KUKA KRL program: rob_ok.src, rob_ok.dat

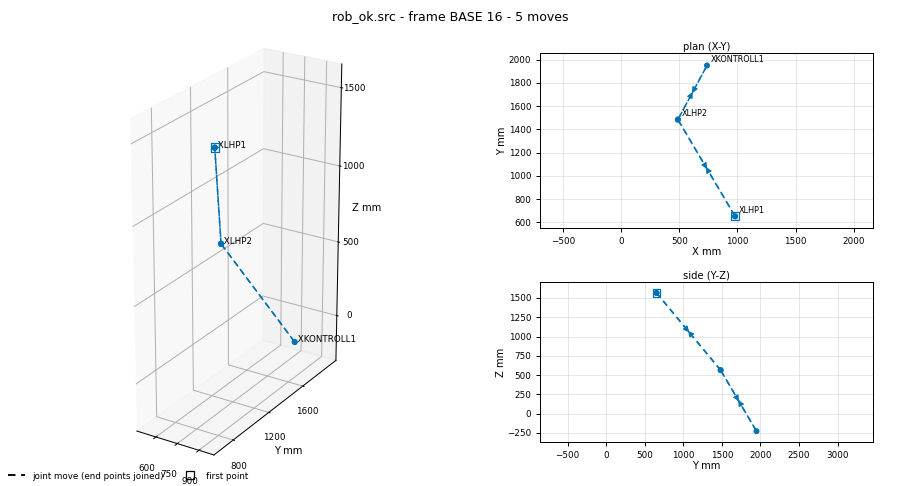
[picture p0: tool path of rob_ok.src in frame BASE 16, 5 of 7 moves have a stored position in this frame; points joined in program order, loops and branches not executed]
--- rob_ok.src ---
&ACCESS RVP
&REL 12
&COMMENT Roboterpruefprogramm
&PARAM TEMPLATE = C:\KRC\ROBOTER\TEMPLATE\VG_HP
&PARAM EDITMASK = *
DEF rob_ok( )
;FOLD INI
;FOLD BASISTECH INI
    GLOBAL INTERRUPT DECL 3 WHEN $STOPMESS==TRUE DO IR_STOPM ( )
    INTERRUPT ON 3
    BAS (#INITMOV,0 )
;ENDFOLD (BASISTECH INI)
;FOLD SPOTTECH INI
    USERSPOT(#INIT)
;ENDFOLD (SPOTTECH INI)
;FOLD GRIPPERTECH INI
    USER_GRP(0,DUMMY,DUMMY,GDEFAULT)
;ENDFOLD (GRIPPERTECH INI)
;FOLD USER INI
;Make your modifications here
;FOLD COLLISION_V_3.01 INI ;%{E}
    IF (COLLISION_DATA[1].I_NR>0) THEN
    GLOBAL INTERRUPT DECL 21 WHEN $IN[COLLISION_DATA[1].I_NR]==FALSE DO COLLSTOP (1,0 )
    ENDIF
    IF (COLLISION_DATA[2].I_NR>0) THEN
    GLOBAL INTERRUPT DECL 22 WHEN $IN[COLLISION_DATA[2].I_NR]==FALSE DO COLLSTOP (2,0 )
    ENDIF
    IF (COLLISION_DATA[3].I_NR>0) THEN
    GLOBAL INTERRUPT DECL 23 WHEN $IN[COLLISION_DATA[3].I_NR]==FALSE DO COLLSTOP (3,0 )
    ENDIF
    IF (COLLISION_DATA[4].I_NR>0) THEN
    GLOBAL INTERRUPT DECL 24 WHEN $IN[COLLISION_DATA[4].I_NR]==FALSE DO COLLSTOP (4,0 )
    ENDIF
;ENDFOLD (Collision)
;ENDFOLD (USER INI)
;ENDFOLD (INI)
;FOLD ; Anlagenbezeichn:               Stations-Nr:;%{PE}%R 5.2.7,%MKUKATPBASIS,%CCOMMENT,%VNORMAL,%P 2:Anlagenbezeichn:               Stations-Nr:
;ENDFOLD
;FOLD ; Stand / Version:;%{PE}%R 5.2.7,%MKUKATPBASIS,%CCOMMENT,%VNORMAL,%P 2:Stand / Version:
;ENDFOLD
;FOLD ; Name Bearbeiter:;%{PE}%R 5.2.7,%MKUKATPBASIS,%CCOMMENT,%VNORMAL,%P 2:Name Bearbeiter:
;ENDFOLD
;Sicherheitsfrage (nur im Musterprogramm, nach teachen entfernen)
wait for false
;FOLD ; ***************************************;%{PE}%R 2.4.6,%MKUKATPBASIS,%CCOMMENT,%VNORMAL,%P 2:***************************************
;ENDFOLD
;FOLD ; A C H T U N G  ! ! !   Nur in T1 fahren;%{PE}%R 2.4.6,%MKUKATPBASIS,%CCOMMENT,%VNORMAL,%P 2:A C H T U N G  ! ! !   Nur in T1 fahren
;ENDFOLD
;FOLD ; ***************************************;%{PE}%R 2.4.6,%MKUKATPBASIS,%CCOMMENT,%VNORMAL,%P 2:***************************************
;ENDFOLD
WAIT FOR $T1
;FOLD PTP HOME  Vel= 100 % DEFAULT;%{PE}%R 3.2.43,%MKUKATPBASIS,%CMOVE,%VPTP,%P 1:PTP, 2:HOME, 3:, 5:100, 7:DEFAULT
    $BWDSTART = FALSE
    PDAT_ACT=PDEFAULT
    BAS(#PTP_DAT)
    FDAT_ACT=FHOME
    BAS(#FRAMES)
    BAS(#VEL_PTP,100)
    $H_POS=XHOME
    PTP XHOME
;ENDFOLD
; PTP ... zur Kontrollposition Roboter teachen
;FOLD PTP LHP1  Vel= 100 % PDAT Tool[16] Base[16];%{PE}%R 3.2.43,%MKUKATPBASIS,%CMOVE,%VPTP,%P 1:PTP, 2:LHP1, 3:, 5:100, 7:PDAT
    $BWDSTART = FALSE
    PDAT_ACT=PPDAT
    BAS(#PTP_DAT)
    FDAT_ACT=FLHP1
    BAS(#FRAMES)
    BAS(#VEL_PTP,100)
    PTP XLHP1
;ENDFOLD
;FOLD PTP LHP2  Vel= 100 % PDAT Tool[16] Base[16];%{PE}%R 3.2.43,%MKUKATPBASIS,%CMOVE,%VPTP,%P 1:PTP, 2:LHP2, 3:, 5:100, 7:PDAT
    $BWDSTART = FALSE
    PDAT_ACT=PPDAT
    BAS(#PTP_DAT)
    FDAT_ACT=FLHP2
    BAS(#FRAMES)
    BAS(#VEL_PTP,100)
    PTP XLHP2
;ENDFOLD
;FOLD ; *********************************************************;%{PE}%R 2.4.6,%MKUKATPBASIS,%CCOMMENT,%VNORMAL,%P 2:*********************************************************
;ENDFOLD
;FOLD ; A C H T U N G  ! ! !   Spitze am IR Flansch befestigen   ;%{PE}%R 2.4.6,%MKUKATPBASIS,%CCOMMENT,%VNORMAL,%P 2:A C H T U N G  ! ! !   Spitze am IR Flansch befestigen
;ENDFOLD
;FOLD ; *********************************************************;%{PE}%R 2.4.6,%MKUKATPBASIS,%CCOMMENT,%VNORMAL,%P 2:*********************************************************
;ENDFOLD
;Spitze am Flansch 02.3 und 03.1
;Spitze an Vorrichtung 01.2 und 03.1
WAIT FOR  $IN[1026]==TRUE
;FOLD ; 1.Kontrollposition;%{PE}%R 2.4.6,%MKUKATPBASIS,%CCOMMENT,%VNORMAL,%P 2:1.Kontrollposition
;ENDFOLD
;FOLD ; Pruefspitze - Roboterflansch         ;%{PE}%R 2.4.6,%MKUKATPBASIS,%CCOMMENT,%VNORMAL,%P 2: Pruefspitze - Roboterflansch
;ENDFOLD
;FOLD ; mit 02.3 03.1 Laenge;%{PE}%R 5.2.17,%MKUKATPBASIS,%CCOMMENT,%VNORMAL,%P 2:mit 02.3 03.1 Laenge
;ENDFOLD
;FOLD PTP KONTROLL1  Vel= 100 % PDAT Tool[16] Base[16];%{PE}%R 3.2.43,%MKUKATPBASIS,%CMOVE,%VPTP,%P 1:PTP, 2:KONTROLL1, 3:, 5:100, 7:PDAT
    $BWDSTART = FALSE
    PDAT_ACT=PPDAT
    BAS(#PTP_DAT)
    FDAT_ACT=FKONTROLL1
    BAS(#FRAMES)
    BAS(#VEL_PTP,100)
    PTP XKONTROLL1
;ENDFOLD
WAIT FOR  $IN[1026]==TRUE ; Kontrollposition IR
;FOLD PTP LHP3  Vel= 100 % PDAT Tool[16] Base[16];%{PE}%R 3.2.43,%MKUKATPBASIS,%CMOVE,%VPTP,%P 1:PTP, 2:LHP3, 3:, 5:100, 7:PDAT
    $BWDSTART = FALSE
    PDAT_ACT=PPDAT
    BAS(#PTP_DAT)
    FDAT_ACT=FLHP3
    BAS(#FRAMES)
    BAS(#VEL_PTP,100)
    PTP XLHP3
;ENDFOLD
;FOLD ; *******************************************************;%{PE}%R 2.4.6,%MKUKATPBASIS,%CCOMMENT,%VNORMAL,%P 2:*******************************************************
;ENDFOLD
;FOLD ; A C H T U N G  ! ! !   Messpitze am IR  entfernen;%{PE}%R 2.4.6,%MKUKATPBASIS,%CCOMMENT,%VNORMAL,%P 2:A C H T U N G  ! ! !   Messpitze am IR  entferne
;ENDFOLD
;FOLD ; *******************************************************;%{PE}%R 2.4.6,%MKUKATPBASIS,%CCOMMENT,%VNORMAL,%P 2:*******************************************************
;ENDFOLD
WAIT FOR  $IN[1026]==TRUE
;FOLD PTP LHP5  Vel= 100 % PDAT Tool[16] Base[16];%{PE}%R 3.2.43,%MKUKATPBASIS,%CMOVE,%VPTP,%P 1:PTP, 2:LHP5, 3:, 5:100, 7:PDAT
    $BWDSTART = FALSE
    PDAT_ACT=PPDAT
    BAS(#PTP_DAT)
    FDAT_ACT=FLHP5
    BAS(#FRAMES)
    BAS(#VEL_PTP,100)
    PTP XLHP5
;ENDFOLD
;FOLD PTP HOME  Vel= 100 % DEFAULT;%{PE}%R 3.2.43,%MKUKATPBASIS,%CMOVE,%VPTP,%P 1:PTP, 2:HOME, 3:, 5:100, 7:DEFAULT
    $BWDSTART = FALSE
    PDAT_ACT=PDEFAULT
    BAS(#PTP_DAT)
    FDAT_ACT=FHOME
    BAS(#FRAMES)
    BAS(#VEL_PTP,100)
    $H_POS=XHOME
    PTP XHOME
;ENDFOLD
END

--- rob_ok.dat ---
&ACCESS RVP
&REL 12
&COMMENT Roboterpruefprogramm
&PARAM TEMPLATE = C:\KRC\ROBOTER\TEMPLATE\VG_HP
&PARAM EDITMASK = *
DEFDAT  ROB_OK
;FOLD EXTERNAL DECLARATIONS;%{PE}%V3.2.0,%MKUKATPBASIS,%CEXT,%VCOMMON,%P
;ENDFOLD


DECL BASIS_SUGG_T LAST_BASIS={POINT1[] "P0                      ",POINT2[] "P0                      ",CP_PARAMS[] "CPDAT0                  ",PTP_PARAMS[] "PDAT0                  ",CONT[] "                        ",CP_VEL[] "2                       ",PTP_VEL[] "100                     "}
DECL E6POS XLHP1={x 980.162,y 652.3817,z 1564.854,a 159.7475,b -4.016941,c 179.1242,s 18,t 43,e1 -100.6665,e2 0.0,e3 0.0,e4 0.0,e5 0.0,e6 0.0}
DECL E6POS XLHP2={x 488.2726,y 1483.844,z 564.0757,a -68.44714,b -8.321163,c -174.3943,s 18,t 3,e1 -100.6665,e2 0.0,e3 0.0,e4 0.0,e5 0.0,e6 0.0}
DECL E6POS XKONTROLL1={x 738.4349,y 1948.431,z -227.0883,a -75.75555,b 7.634907,c -102.5782,s 18,t 35,e1 -100.6661,e2 0.0,e3 0.0,e4 0.0,e5 0.0,e6 0.0}
DECL E6POS XLHP3={x 488.2894,y 1483.862,z 564.086,a -68.44775,b -8.320516,c -174.3938,s 18,t 3,e1 -100.6661,e2 0.0,e3 0.0,e4 0.0,e5 0.0,e6 0.0}
DECL E6POS XLHP5={x 980.1634,y 652.3851,z 1564.827,a 159.7478,b -4.017778,c 179.1253,s 18,t 43,e1 -100.6665,e2 0.0,e3 0.0,e4 0.0,e5 0.0,e6 0.0}
DECL FDAT FLHP1={TOOL_NO 16,BASE_NO 16,IPO_FRAME #BASE}
DECL FDAT FLHP2={TOOL_NO 16,BASE_NO 16,IPO_FRAME #BASE}
DECL FDAT FKONTROLL1={TOOL_NO 16,BASE_NO 16,IPO_FRAME #BASE}
DECL FDAT FLHP3={TOOL_NO 16,BASE_NO 16,IPO_FRAME #BASE}
DECL FDAT FLHP5={TOOL_NO 16,BASE_NO 16,IPO_FRAME #BASE}
DECL FDAT FHOME={TOOL_NO 1,BASE_NO 0,IPO_FRAME #BASE}
DECL PDAT PPDAT={VEL 100.0,ACC 100.0,APO_DIST 100.0}
ENDDAT
